# B&R Automation Studio project AutoConTest
Automation Studio 6.1.1.14; technology packages: OpcUaCs 6.0.0

## Configuration Config1

CPU X20CP1684, AutomationRuntime 6.0.2, Build 11.3.0, Vc 6.0.0

### Task classes (Cpu.sw)
```
Cyclic#4:
  Program <- Program.prg
```

### Hardware
```
X20CP1684 : X20CP1684 v1.8.1.0
  FileDevice1
  FileDeviceName1 = USER
  FileDevicePath1 = USER_PATH
```

## Logical view

Binary libraries used (declarations not repeated): operator, runtime, AsIecCon, astime


### Program Logical/Program (IEC)

#### Variables.var
```iecst
VAR
	input : BOOL;
	output : BOOL;
END_VAR
```

#### Cyclic.ld
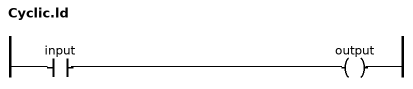
Diagram, in the editor's own instruction-list form stored in the file:
```il
PROGRAM _CYCLIC

{NetworkNumber := 1}
LD	input
ST	output

END_PROGRAM
```

#### Exit.ld
Diagram, in the editor's own instruction-list form stored in the file:
```il
PROGRAM _EXIT

END_PROGRAM
```

#### Init.ld
Diagram, in the editor's own instruction-list form stored in the file:
```il
PROGRAM _INIT

END_PROGRAM
```

Listed in the project but not available here: Logical/Global.typ, Logical/Global.var
